// TIA Portal V20 export
DATA_BLOCK "TestVarIdent"   // DB76
TITLE = Test tags fuer ident / Test tags for ident
AUTHOR : SICAR
FAMILY : Ident
VERSION : 1.0
// Test tags fuer ident / Test tags for ident
// stored: MemoryReserve 100
   VAR
      init1 : Bool := FALSE;   // Init 1
      read1 : Bool := FALSE;   // Read1
      write1 : Bool := FALSE;   // Write1
      init2 : Bool := FALSE;   // Init 2
      read2 : Bool := FALSE;   // Read2
      write2 : Bool := FALSE;   // Write2
      testString : String[32] := '';   // Test string
      charArr : Array[1..32] of Byte;   // Array of characters / Character Array
      prgNoMan : USInt := 0;   // Progrmm Nummer schreiben manual / Program number manual
      enableManCtrlRf : Bool := FALSE;   // Freigabe Manual Steuerung / Enable manual control RFID
      enableOption : Bool := FALSE;   // Freiegbae Optionen / Enable options
      enableManCtrlMV : Bool := FALSE;   // Enable manual control MV
   END_VAR
BEGIN
   charArr[1..32] := 16#00;
END_DATA_BLOCK
